// TwinCAT 3 PLC project FactoryIOLibrary
// Title: FactoryIO_Library
// Company: Privat
// Author: Entwickler
// ProjectVersion: 0.0.8
// Description: This library contains function blocks to control scenes in FactoryIO.
// ProgramVersion: 3.1.4026.24
// libraries:
//   Tc2_Standard, * (Beckhoff Automation GmbH)
//   Tc2_System, * (Beckhoff Automation GmbH)
//   Tc2_Utilities, * (Beckhoff Automation GmbH)
//   Tc3_Module, * (Beckhoff Automation GmbH)
// project tree:
//   DUTs/Communication/ADS/ ADSCommunicationInterface.TcDUT
//   DUTs/HMI/Header/ HMIHeader.TcDUT (not stored)
//   DUTs/HMI/MachineSection/ HMIMovementForkInterface.TcDUT, HMIMovementInterface.TcDUT, HMIRFIDControlInterface.TcDUT, HMIRFIDDataInterface.TcDUT, HMIRFIDInterface.TcDUT, HMIRFIDStatusInterface.TcDUT (not stored), HMIRuncontrolInterface.TcDUT, HMIWindowSwitch.TcDUT (not stored), HMIWorkpieceInterface.TcDUT (not stored), MachineSection.TcDUT (not stored), MachineSectionHMIInterface.TcDUT
//   DUTs/HMI/NumericalInput/ HMIButtonNumericalInputInterface.TcDUT (not stored), HMINumericalInputInterface.TcDUT, HMINumericalInputLineInterface.TcDUT (not stored)
//   DUTs/HMI/SettingLine/ HMIButtonSettingLineInterface.TcDUT (not stored), HMISettingLineInterface.TcDUT (not stored)
//   DUTs/OperatingMode/ ActionState.TcDUT (not stored), FaultWarningState.TcDUT, HMIActionState.TcDUT (not stored), HMIInterfaceOperatingMode.TcDUT, HMIToPLCOperatingMode.TcDUT, OperatingMode.TcDUT, OperatingModeHomeing.TcDUT (not stored), PLCToHMIOperatingMode.TcDUT
//   DUTs/PickPlace/ PickPlacePosition.TcDUT (not stored)
//   DUTs/PositingBar/ PositingBarAlignmentDirection.TcDUT
//   DUTs/RFID/ RFIDReadSerialnumberStates.TcDUT (not stored), RFIDReadWriteDataStates.TcDUT
//   DUTs/VisionSensor/ VisionSensorParttype.TcDUT
//   POUs/AnalogValueHandling/ FC_AnalogInputValueHandling.TcPOU (not stored), FC_AnalogOutputValueHandling.TcPOU
//   POUs/Aufzug/ FB_Elevator.TcPOU (not stored)
//   POUs/Communication/ADS/ FB_ADSCommunicationStatus.TcPOU
//   POUs/Emitter/ FB_Emitter.TcPOU (not stored)
//   POUs/Foerderband/ FB_Foerderband.TcPOU
//   POUs/HMI/ FB_HMIHeader.TcPOU, FC_InitializingSettingLines.TcPOU (not stored)
//   POUs/OperatingMode/ FB_OperatingMode.TcPOU
//   POUs/PickPlace/ FB_PickPlace_DigitalAnalog.TcPOU (not stored)
//   POUs/PositingBar/ FB_PositingBar.TcPOU (not stored)
//   POUs/Remover/ FB_Remover.TcPOU
//   POUs/RFID/ FB_RFID.TcPOU (not stored)
//   POUs/VisionSensor/ FB_VisionSensor.TcPOU (not stored)
//   POUs/Warehouse/ FB_StackerCrane_Analog.TcPOU, FB_StackerCrane_Numerical.TcPOU
//   Version/ Global_Version.TcGVL

// ---- DUTs/Communication/ADS/ADSCommunicationInterface.TcDUT
TYPE ADSCommunicationInterface :
STRUCT
	LocalAMSNetId	:	STRING;
	DeviceIpAddress	:	STRING;
	RuntimeStatus	:	STRING;
	HeartbeatPLC	:	BOOL;
	HeartbeatHMI	:	BOOL;
END_STRUCT
END_TYPE

// ---- DUTs/HMI/MachineSection/HMIMovementForkInterface.TcDUT
TYPE HMIMovementForkInterface :
STRUCT
	ForkMovementSettingLines	:	ARRAY [1..3] of HMISettingLineInterface;
END_STRUCT
END_TYPE

// ---- DUTs/HMI/MachineSection/HMIMovementInterface.TcDUT
TYPE HMIMovementInterface :
STRUCT
	MovementSettingLines	:	ARRAY [1..3] OF HMISettingLineInterface;
	NumericalInput	:	HMINumericalInputInterface;
END_STRUCT
END_TYPE

// ---- DUTs/HMI/MachineSection/HMIRFIDControlInterface.TcDUT
TYPE HMIRFIDControlInterface :
STRUCT
	ExecuteCommand	:	BOOL;
	SelectedCommand	:	WORD;
	SelectedMemoryIndex	:	WORD;
END_STRUCT
END_TYPE

// ---- DUTs/HMI/MachineSection/HMIRFIDDataInterface.TcDUT
TYPE HMIRFIDDataInterface :
STRUCT
	SingleReadValue	:	WORD;
	SingleWriteValue	:	WORD;
	AllReadData	:	ARRAY[0..127] OF WORD;
	AllWriteData	:	ARRAY[0..127] OF WORD;
END_STRUCT
END_TYPE

// ---- DUTs/HMI/MachineSection/HMIRFIDInterface.TcDUT
TYPE HMIRFIDInterface :
STRUCT
	RFIDStatus	:	HMIRFIDStatusInterface;
	RFIDControl	:	HMIRFIDControlInterface;
	RFIDData	:	HMIRFIDDataInterface;
END_STRUCT
END_TYPE

// ---- DUTs/HMI/MachineSection/HMIRuncontrolInterface.TcDUT
TYPE HMIRuncontrolInterface :
STRUCT
	RuncontrolSettingLines	:	ARRAY [1..3] of HMISettingLineInterface;
END_STRUCT
END_TYPE

// ---- DUTs/HMI/MachineSection/MachineSectionHMIInterface.TcDUT
TYPE MachineSectionHMIInterface :
STRUCT
	ActiveMachineSection : MachineSection;
	SelectedActor : INT;
	Movements : HMIMovementInterface;
	Forks : HMIMovementForkInterface;
	Runcontrols : HMIRuncontrolInterface;
	RFID : HMIRFIDInterface;
	Workpiece : HMIWorkpieceInterface;
END_STRUCT
END_TYPE

// ---- DUTs/HMI/NumericalInput/HMINumericalInputInterface.TcDUT
TYPE HMINumericalInputInterface :
STRUCT
	CaptionNumericalInput	:	STRING;
	IsVisibleNumericalInput	:	BOOL;
	ValueLinesNumericalInput	:	ARRAY[1..2] OF HMINumericalInputLineInterface;
	ButtonsNumericalInput	:	ARRAY[1..2] OF HMIButtonNumericalInputInterface;
END_STRUCT
END_TYPE

// ---- DUTs/OperatingMode/FaultWarningState.TcDUT
TYPE FaultWarningState :
STRUCT
	IsActive :	BOOL;
END_STRUCT
END_TYPE

// ---- DUTs/OperatingMode/HMIInterfaceOperatingMode.TcDUT
TYPE HMIInterfaceOperatingMode :
STRUCT
	PLCToHMI	:	PLCToHMIOperatingMode;
	HMIToPLC	:	HMIToPLCOperatingMode;
END_STRUCT
END_TYPE

// ---- DUTs/OperatingMode/HMIToPLCOperatingMode.TcDUT
TYPE HMIToPLCOperatingMode :
STRUCT
	Manuel	:	HMIActionState;
	Automatic	:	HMIActionState;
	AutomaticStart	:	HMIActionState;
	AutomaticStop	:	HMIActionState;
	AutomaticHome	:	HMIActionState;
	Quit	:	HMIActionState;
	Reset	:	HMIActionState;
END_STRUCT
END_TYPE

// ---- DUTs/OperatingMode/OperatingMode.TcDUT
TYPE OperatingMode :
STRUCT
	ManuelIsActive	:	BOOL;
	AutomaticIsActive	:	BOOL;
	EStop			:	ActionState;
	Fault			:	FaultWarningState;
	Warning			:	FaultWarningState;
	AutomaticStart	:	ActionState;
	AutomaticStop	:	ActionState;
	Reset	:	ActionState;
	Quit	:	ActionState;
	AutomaticHome	:	OperatingModeHomeing;
END_STRUCT
END_TYPE

// ---- DUTs/OperatingMode/PLCToHMIOperatingMode.TcDUT
TYPE PLCToHMIOperatingMode :
STRUCT
	Manuel	:	ActionState;
	Automatic	:	ActionState;
	AutomaticStart	:	ActionState;
	Automaticstop	:	ActionState;
	AutomaticHome	:	ActionState;
	Reset	:	ActionState;
	Quit	:	ActionState;
	Fault	:	ActionState;
	
END_STRUCT
END_TYPE

// ---- DUTs/PositingBar/PositingBarAlignmentDirection.TcDUT
{attribute 'qualified_only'}
{attribute 'strict'}
{attribute 'to_string'}
TYPE PositingBarAlignmentDirection :
(
	AlingmentLeft := 0,
	AlingmentRight
);
END_TYPE

// ---- DUTs/RFID/RFIDReadWriteDataStates.TcDUT
{attribute 'qualified_only'}
{attribute 'strict'}
{attribute 'to_string'}
TYPE RFIDReadWriteDataStates :
(
	WAITINGTRIGGER := 0,
	SETTRIGGER,
	WAITINGRESPONSE,
	RESPONSE,
	ERRORACTIVE,
	FINISHED
);
END_TYPE

// ---- DUTs/VisionSensor/VisionSensorParttype.TcDUT
{attribute 'qualified_only'}
{attribute 'strict'}
{attribute 'to_string'}
TYPE VisionSensorParttype :
(
	None := 0,
	BlueRawMaterial,
	BlueProductLid,
	BlueProductBase,
	GreenRawMaterial,
	GreenProductLid,
	GreenProductBase,
	MetalRawMaterial,
	MetalProductLid,
	MetalProductBase,
	NotDectedable := 100
);
END_TYPE

// ---- Version/Global_Version.TcGVL
{attribute 'TcGenerated'}
{attribute 'no-analysis'}
{attribute 'linkalways'}
// This function has been automatically generated from the project information.
VAR_GLOBAL CONSTANT
	{attribute 'const_non_replaced'}
	stLibVersion_FactoryIO_Library : ST_LibVersion := (iMajor := 0, iMinor := 0, iBuild := 8, iRevision := 0, nFlags := 0, sVersion := '0.0.8');
END_VAR

// ---- POUs/AnalogValueHandling/FC_AnalogOutputValueHandling.TcPOU
FUNCTION FC_AnalogOutputValueHandling
VAR_INPUT
	Setpoint	:	REAL;
	UpperLimit	:	REAL;
	LowerLimit	:	REAL;
END_VAR
VAR_OUTPUT
	ConvertedValue	:	WORD;
END_VAR
VAR
	tempCalculatedValue	:	REAL;
	tempConvertedValue	:	WORD;
	tempValueWithOffset	:	WORD;
END_VAR

tempCalculatedValue := Setpoint * 10.0/(UpperLimit - LowerLimit);
tempConvertedValue := TO_WORD(tempCalculatedValue * 10.0);
tempValueWithOffset := tempConvertedValue * 10;

ConvertedValue := tempValueWithOffset;

END_FUNCTION

// ---- POUs/Communication/ADS/FB_ADSCommunicationStatus.TcPOU
FUNCTION_BLOCK FB_ADSCommunicationStatus
VAR_INPUT
	Timeout	:	TIME := T#1S;
	TimeoutHMI	:	TIME := T#1S;
	LocalAdsPort	:	T_AmsPort := 851;
	HeartbeatHMI	:	BOOL;
END_VAR
VAR
	instReadLocalAMSNetId	:	FB_GetLocalAmsNetId;
	statExecuteReadingLocalAMSNetId	:	BOOL := TRUE;
	statBusyReadLocalAMSNetId	:	BOOL;
	statErrorReadLocalAMSNetId	:	BOOL;
	statErrorNumberReadLocalAMSNetId	:	UDINT;
	statReadLocalAMSNetId	:	T_AmsNetID;
	statReadLocalAMSNetIdSeprated	:	T_AmsNetIdArr;
	
	statGettingIpAddress	:	BOOL;
	statLocalIpAddress	:	STRING;
	
	instReadADSState	:	ADSRDSTATE;
	statExecuteReadingAdsState	:	BOOL;
	statBusyReadAdsState	:	BOOL;
	statErrorReadAdsState	:	BOOL;
	statErrorNumberAdsState	:	UDINT;
	statReadAdsState	:	UDINT;
	
	statConvertingAdsState	:	BOOL;
	statConvertedAdsState	:	STRING;
	
	instHearbeatEvaluationHMITrue	:	TON;
	instHearbeatEvaluationHMIFalse	:	TON;
	statErrorHeartbeatHMIToLongTrue	:	BOOL;
	statErrorHeartbeatHMIToLongFalse	:	BOOL;
	statHearbeatHMIIsKeepAlive	:	BOOL;
	
	instHearbeatPLCTrue	:	TON;
	statHeartbeatPLCTrue	:	BOOL;
	statHearbeatPLC	:	BOOL;
END_VAR

(*===================== Reading local AMSNetId =====================*)
instReadLocalAMSNetId(bExecute := statExecuteReadingLocalAMSNetId,
					  tTimeOut := Timeout,
					  bBusy => statBusyReadLocalAMSNetId,
					  bError => statErrorReadLocalAMSNetId,
					  nErrId => statErrorNumberReadLocalAMSNetId,
					  AddrString => statReadLocalAMSNetId,
					  AddrBytes => statReadLocalAMSNetIdSeprated);
					  
IF NOT statBusyReadLocalAMSNetId AND NOT statErrorReadLocalAMSNetId AND
	statExecuteReadingLocalAMSNetId THEN
	statExecuteReadingLocalAMSNetId := FALSE;
	statGettingIpAddress := TRUE;
	statExecuteReadingAdsState := TRUE;
END_IF

(*===================== Getting IP-Address =====================*)
IF statGettingIpAddress THEN
	statLocalIpAddress := GetDeviceIpAddress(statReadLocalAMSNetIdSeprated);
	statGettingIpAddress := FALSE;
END_IF

(*===================== Reading Ads state =====================*)
instReadADSState(NETID := statReadLocalAMSNetId,
				 PORT := LocalAdsPort,
				 RDSTATE := statExecuteReadingAdsState,
			     TMOUT := Timeout,
				 BUSY => statBusyReadAdsState,
				 ERR => statErrorReadAdsState,
				 ERRID => statErrorNumberAdsState,
				 ADSSTATE => statReadAdsState);
					  
IF NOT statBusyReadAdsState AND NOT statErrorReadAdsState AND
	statExecuteReadingAdsState THEN
	statExecuteReadingAdsState := FALSE;
	statConvertingAdsState := TRUE;
END_IF

(*===================== Converting Ads state =====================*)
IF statConvertingAdsState THEN
	statConvertedAdsState := ConvertRuntimestatusInString(statReadAdsState);
	statConvertingAdsState := FALSE;
END_IF

(*===================== Evaluating Heartbeat HMI =====================*)
instHearbeatEvaluationHMITrue(IN := HeartbeatHMI,
							  PT := TimeoutHMI,
							  Q => statErrorHeartbeatHMIToLongTrue);
instHearbeatEvaluationHMIFalse(IN := NOT HeartbeatHMI,
							  PT := TimeoutHMI,
							  Q => statErrorHeartbeatHMIToLongFalse);
							  

statHearbeatHMIIsKeepAlive := NOT statErrorHeartbeatHMIToLongTrue AND NOT statErrorHeartbeatHMIToLongFalse;

(*===================== Creating Heartbeat PLC =====================*)
instHearbeatPLCTrue(IN := NOT statHeartbeatPLCTrue,
					PT := TimeoutHMI,
					Q => statHeartbeatPLCTrue);
							  
IF statHeartbeatPLCTrue THEN
	statHearbeatPLC := NOT statHearbeatPLC;
END_IF

PROPERTY PUBLIC AdsState : String
GET
AdsState := statConvertedAdsState;
END_GET
END_PROPERTY

METHOD PRIVATE ConvertRuntimestatusInString : String
VAR_INPUT
	CurrentDeviceStatus 	: 	UDINT;
END_VAR
VAR
	tempConvertedDeviceStatus	:	STRING;
END_VAR
CASE CurrentDeviceStatus OF
	0:
		tempConvertedDeviceStatus := 'Invalid';
	1:
		tempConvertedDeviceStatus := 'Idle';
	2:
		tempConvertedDeviceStatus := 'Reset';
	3:
		tempConvertedDeviceStatus := 'Init';
	4:
		tempConvertedDeviceStatus := 'Start';
	5:
		tempConvertedDeviceStatus := 'Run';
	6:
		tempConvertedDeviceStatus := 'Stop';
	7:
		tempConvertedDeviceStatus := 'Save cfg';
	8:
		tempConvertedDeviceStatus := 'Load cfg';
	9:
		tempConvertedDeviceStatus := 'Power failure';
	10:
		tempConvertedDeviceStatus := 'Power good';
	11:
		tempConvertedDeviceStatus := 'Error';
	12:
		tempConvertedDeviceStatus := 'Shutdown';
	13:
		tempConvertedDeviceStatus := 'Suspend';
	14:
		tempConvertedDeviceStatus := 'Resume';
	15:
		tempConvertedDeviceStatus := 'Config';
	16:
		tempConvertedDeviceStatus := 'Reconfig';
	17:
		tempConvertedDeviceStatus := 'Stopping';
	18:
		tempConvertedDeviceStatus := 'Incompatible';
	19:
		tempConvertedDeviceStatus := 'Execption';
	ELSE
		tempConvertedDeviceStatus := 'Not defined in system';			
END_CASE

ConvertRuntimestatusInString := tempConvertedDeviceStatus;
END_METHOD

METHOD PRIVATE GetDeviceIpAddress : String
VAR_INPUT
	CurrentAMSNetId	:	T_AmsNetIdArr;
END_VAR
VAR
	tempRunCounter	:	INT;
	tempIpAddressConverted	:	STRING;
END_VAR
FOR tempRunCounter := 0 TO 3 DO
	tempIpAddressConverted := CONCAT(tempIpAddressConverted, BYTE_TO_STRING(CurrentAMSNetId[tempRunCounter]));
	IF tempRunCounter < 3 THEN
		tempIpAddressConverted := CONCAT(tempIpAddressConverted, '.');
	END_IF
END_FOR

GetDeviceIpAddress := tempIpAddressConverted;
END_METHOD

PROPERTY PUBLIC HMICommunicationIsActive : BOOL
GET
HMICommunicationIsActive := statHearbeatHMIIsKeepAlive;
END_GET
END_PROPERTY

PROPERTY PUBLIC LocalAMSNetId : String
GET
LocalAMSNetId := statReadLocalAMSNetId;
END_GET
END_PROPERTY

PROPERTY PUBLIC LocalIpAddress : String
GET
LocalIpAddress := statLocalIpAddress;
END_GET
END_PROPERTY

PROPERTY PUBLIC PLCHeartbeatHMICommunication : BOOL
GET
PLCHeartbeatHMICommunication := statHearbeatPLC;
END_GET
END_PROPERTY

END_FUNCTION_BLOCK

// ---- POUs/Foerderband/FB_Foerderband.TcPOU
FUNCTION_BLOCK FB_Foerderband
VAR_INPUT
	SensorInfeed	:	BOOL;	//Sensor am Band Einlauf
	SensorOutfeed	:	BOOL;	//Sensor am Band Auslauf
	MaximumTimeRuncontrol	:	TIME;	//Maximale Zeit bis Fehler Laufkontrolle aktiviert wird
END_VAR
VAR_OUTPUT
	MotorForward	:	BOOL;	//Motor vorwaerts drehen
	MotorBackward	:	BOOL;	//Motor rueckwaerts drehen
	RuncontrolForwardActive	:	BOOL;	//Laufkontrolle in Vorwaerts-Richtung aktiv
	RuncontrolBackwardActive	:	BOOL;	//Laufkontrolle in Rueckwaerts-Richtung aktiv
	Error	:	BOOL;	//Fehler aktiv
END_VAR
VAR_IN_OUT
	OperatingMode	:	OperatingMode;	//Schnittstelle für Betriebsarten
END_VAR
VAR
	statMotorForward	:	BOOL;
	statMotorBackward	:	BOOL;
	statRuncontrolForward	:	BOOL;
	statRuncontrolBackward	:	BOOL;
	statErrorRuncontrolForward	:	BOOL;
	statErrorRuncontrolBackward	:	BOOL;
	statTimeRuncontrolForward	:	TON;
	statTimeRuncontrolBackward	:	TON;
END_VAR

(*===================== Motor Forward =====================*)
statMotorForward := statMotorForward AND OperatingMode.AutomaticIsActive
									 AND(OperatingMode.AutomaticStart.IsActive OR 
										 OperatingMode.AutomaticHome.IsActive) AND NOT
										 statMotorBackward AND NOT
									 	 OperatingMode.AutomaticStop.IsActive AND NOT
									 	 OperatingMode.EStop.IsActive AND NOT
										 statErrorRuncontrolForward;
(*===================== Motor Backward =====================*)
statMotorBackward := statMotorBackward AND OperatingMode.AutomaticIsActive
									   AND(OperatingMode.AutomaticStart.IsActive OR 
										   OperatingMode.AutomaticHome.IsActive) AND NOT
										   statMotorForward AND NOT
									 	   OperatingMode.AutomaticStop.IsActive AND NOT
									 	   OperatingMode.EStop.IsActive AND NOT
										   statErrorRuncontrolBackward;
(*===================== Runcontrol Forward =====================*)
IF statMotorForward AND NOT statRuncontrolForward THEN
	statRuncontrolForward := TRUE;
ELSIF (statRuncontrolForward AND SensorOutfeed) OR
	(OperatingMode.Reset.IsActive AND statErrorRuncontrolForward)
THEN
		statRuncontrolForward := FALSE;
END_IF

statTimeRuncontrolForward(IN:= statRuncontrolForward,
						  PT:= MaximumTimeRuncontrol);
IF OperatingMode.Quit.IsActive THEN
	statErrorRuncontrolForward := FALSE;
END_IF
IF statTimeRuncontrolForward.Q THEN
	statErrorRuncontrolForward := TRUE;
END_IF
(*===================== Runcontrol Backward =====================*)
IF statMotorBackward AND NOT statRuncontrolBackward THEN
	statRuncontrolBackward := TRUE;
ELSIF statRuncontrolBackward AND SensorInfeed OR
	(OperatingMode.Reset.IsActive AND statErrorRuncontrolBackward)
THEN
		statRuncontrolBackward := FALSE;
END_IF

statTimeRuncontrolBackward(IN:= statRuncontrolBackward,
						   PT:= MaximumTimeRuncontrol);
IF OperatingMode.Quit.IsActive THEN
	statErrorRuncontrolBackward := FALSE;
END_IF
IF statTimeRuncontrolBackward.Q THEN
	statErrorRuncontrolBackward := TRUE;
END_IF
(*===================== Outputs =====================*)
MotorForward := statMotorForward;
MotorBackward := statMotorBackward;
RuncontrolForwardActive := statRuncontrolForward;
RuncontrolBackwardActive := statRuncontrolBackward;
Error := statErrorRuncontrolForward OR statErrorRuncontrolBackward;
OperatingMode.Fault.IsActive :=  statErrorRuncontrolForward OR statErrorRuncontrolBackward;

METHOD PUBLIC Motor_Off
VAR_INPUT
	Motor_Stop	:	BOOL;
END_VAR
IF Motor_Stop THEN
	statMotorForward := FALSE;
	statMotorBackward := FALSE;
END_IF
END_METHOD

METHOD MotorBackward_On
VAR_INPUT
	MotorBackward_Start	:	BOOL;
END_VAR
IF OperatingMode.AutomaticIsActive AND
(OperatingMode.AutomaticStart.IsActive OR 
 OperatingMode.AutomaticHome.IsActive) AND NOT
 statMotorForward AND NOT
 OperatingMode.AutomaticStop.IsActive AND NOT
 OperatingMode.EStop.IsActive AND NOT
 statErrorRuncontrolBackward AND NOT
 statMotorBackward AND
 MotorBackward_Start
 THEN
 	statMotorBackward := TRUE;
END_IF
END_METHOD

METHOD PUBLIC MotorForward_On
VAR_INPUT
	MotorForward_Start	:	BOOL;
END_VAR
IF  OperatingMode.AutomaticIsActive AND
(OperatingMode.AutomaticStart.IsActive OR 
 OperatingMode.AutomaticHome.IsActive) AND NOT
 statMotorBackward AND NOT
 OperatingMode.AutomaticStop.IsActive AND NOT
 OperatingMode.EStop.IsActive AND NOT
 statErrorRuncontrolForward AND NOT
 statMotorForward AND
 MotorForward_Start
 THEN
	statMotorForward := TRUE;
END_IF
END_METHOD

END_FUNCTION_BLOCK

// ---- POUs/HMI/FB_HMIHeader.TcPOU
FUNCTION_BLOCK FB_HMIHeader
VAR_INPUT
	NameApplication	:	STRING;
	OperatingModeHMIInterface	:	HMIInterfaceOperatingMode;
END_VAR
VAR_OUTPUT
END_VAR
VAR_IN_OUT
	HeaderHMIInterface	:	HMIHeader;
END_VAR
VAR
	statHeaderHMIInterface	:	HMIHeader;
END_VAR

(*===================== Name Application =====================*)
statHeaderHMIInterface.NameApplication := NameApplication;
(*===================== Name Application =====================*)
statHeaderHMIInterface.ErrorIsActive := OperatingModeHMIInterface.PLCToHMI.Fault.IsActive;
(*===================== Operating Mode =====================*)
IF OperatingModeHMIInterface.PLCToHMI.Manuel.IsActive THEN
	statHeaderHMIInterface.PathOperatingMode := 'Images/Manual_Mode.svg';
	statHeaderHMIInterface.State := 1;
ELSIF OperatingModeHMIInterface.PLCToHMI.Automatic.IsActive THEN
	statHeaderHMIInterface.PathOperatingMode := 'Images/Automatic_Mode.svg';
	statHeaderHMIInterface.State := 2;
END_IF
(*===================== Operating State =====================*)
IF OperatingModeHMIInterface.PLCToHMI.AutomaticStart.IsActive THEN
	statHeaderHMIInterface.PathMachineState := 'Images/Machine_Run.svg';
	statHeaderHMIInterface.State := 3;
ELSIF OperatingModeHMIInterface.PLCToHMI.AutomaticStop.IsActive THEN
	statHeaderHMIInterface.PathMachineState := 'Images/Machine_Stop.svg';
	statHeaderHMIInterface.State := 2;	
ELSIF OperatingModeHMIInterface.PLCToHMI.AutomaticHome.IsActive THEN
	statHeaderHMIInterface.PathMachineState := 'Images/Home-Symbol.svg';
	statHeaderHMIInterface.State := 4;			
END_IF
(*===================== Outputs =====================*)
HeaderHMIInterface := statHeaderHMIInterface;

END_FUNCTION_BLOCK

// ---- POUs/OperatingMode/FB_OperatingMode.TcPOU
FUNCTION_BLOCK FB_OperatingMode
VAR_INPUT
	PermissionHardware	:	BOOL;	//Permission hardware ready for operation
	PermissionSoftware	:	BOOL;	//Permission from safety machine ready for start
	E_Stop	:	BOOL;	//Button E-Stop
	OperatingModeManual	:	BOOL;	//Operating Mode manual is selected
	OperatingModeAutomatic	:	BOOL;	//Operating Mode automatic is selected
END_VAR
VAR_OUTPUT
	LEDStart	:	BOOL;	//Indicator to show state automatic start
	LEDStop	:	BOOL;	//Indicator to show state automatic stop
	LEDHome	:	BOOL;	//Indicator to show state automatic home
	LEDReset	:	BOOL;	//Indicator to show state reset
	LEDQuit	:	BOOL;	//Indicator to show state quit
END_VAR
VAR_IN_OUT
	HMIInterface	:	HMIInterfaceOperatingMode;
END_VAR
VAR
	statRisingEdgeAutomaticActivated	:	BOOL;	//Rising edge, used when Automatic is activated
	statOperatingMode	:	OperatingMode;
	statResetMethod	:	BOOL;
	statQuitMethod	:	BOOL;
	
	statHMIInterface	:	HMIInterfaceOperatingMode;
	statRisingEdgeManuelButtonPressedMachine	:	R_TRIG;
	statRisingEdgeManuelButtonPressedHMI	:	R_TRIG;
	statRisingEdgeAutomaticButtonPressedMachine	:	R_TRIG;
	statRisingEdgeAutomaticButtonPressedHMI	:	R_TRIG;
	statRisingEdgeAutomaticStartButtonPressedHMI	:	R_TRIG;
	statRisingEdgeAutomaticStopButtonPressedHMI	:	R_TRIG;
	statRisingEdgeAutomaticHomeButtonPressedHMI	:	R_TRIG;
END_VAR

(*===================== HMI-Interface umladen =====================*)
statHMIInterface := HMIInterface;
(*===================== Betriebsartenwahl =====================*)
statRisingEdgeManuelButtonPressedMachine(CLK := OperatingModeManual);
statRisingEdgeManuelButtonPressedHMI(CLK := statHMIInterface.HMIToPLC.Manuel.IsSelected);
statRisingEdgeAutomaticButtonPressedMachine(CLK := OperatingModeAutomatic);
statRisingEdgeAutomaticButtonPressedHMI(CLK := statHMIInterface.HMIToPLC.Automatic.IsSelected);
(*===================== Operating Manual =====================*)
statHMIInterface.PLCToHMI.Manuel.PreconditionsFullfilled := TRUE;
IF statRisingEdgeManuelButtonPressedMachine.Q OR
	(statRisingEdgeManuelButtonPressedHMI.Q AND statHMIInterface.PLCToHMI.Manuel.PreconditionsFullfilled)
	THEN
	statOperatingMode.ManuelIsActive := TRUE;
	statOperatingMode.AutomaticIsActive := FALSE;
END_IF
// statOperatingMode.ManuelIsActive := OperatingModeManual; 
(*===================== Operating Automatic =====================*)
statHMIInterface.PLCToHMI.Automatic.PreconditionsFullfilled := TRUE;
// statOperatingMode.AutomaticIsActive := OperatingModeAutomatic;
IF statRisingEdgeAutomaticButtonPressedMachine.Q OR
	(statRisingEdgeAutomaticButtonPressedHMI.Q AND statHMIInterface.PLCToHMI.Manuel.PreconditionsFullfilled)
	THEN
	statOperatingMode.AutomaticIsActive := TRUE;
	statOperatingMode.ManuelIsActive := FALSE;
END_IF
(*===================== HMI-Interface Betriebsarten =====================*)
statHMIInterface.PLCToHMI.Automatic.IsActive := statOperatingMode.AutomaticIsActive; 
statHMIInterface.PLCToHMI.Manuel.IsActive := statOperatingMode.ManuelIsActive;
(*===================== E-Stop is active =====================*)
statOperatingMode.EStop.PreconditionsFullfilled := TRUE;
statOperatingMode.EStop.IsActive := NOT E_Stop AND statOperatingMode.EStop.PreconditionsFullfilled;
(*===================== Reset is active =====================*)
statOperatingMode.Reset.PreconditionsFullfilled := TRUE;
statHMIInterface.PLCToHMI.Reset.PreconditionsFullfilled := statOperatingMode.Reset.PreconditionsFullfilled;
statOperatingMode.Reset.IsActive := (statResetMethod OR
									 statHMIInterface.HMIToPLC.Reset.IsSelected) AND 
									statOperatingMode.Reset.PreconditionsFullfilled;
statHMIInterface.PLCToHMI.Reset.IsActive := statOperatingMode.Reset.IsActive; 
(*===================== Quit is active =====================*)
statOperatingMode.Quit.PreconditionsFullfilled := TRUE;
statHMIInterface.PLCToHMI.Quit.PreconditionsFullfilled := statOperatingMode.Quit.PreconditionsFullfilled; 
statOperatingMode.Quit.IsActive := (statQuitMethod OR
									statHMIInterface.HMIToPLC.Quit.IsSelected) AND 
									statOperatingMode.Quit.PreconditionsFullfilled;
statHMIInterface.PLCToHMI.Quit.IsActive := statOperatingMode.Quit.IsActive; 
(*===================== Automatic Start is active =====================*)
statRisingEdgeAutomaticStartButtonPressedHMI(CLK := statHMIInterface.HMIToPLC.AutomaticStart.IsSelected);
statOperatingMode.AutomaticStart.PreconditionsFullfilled := PermissionHardware AND PermissionSoftware AND
												  			E_Stop AND NOT statOperatingMode.Reset.IsActive AND NOT
												  			statOperatingMode.AutomaticHome.IsActive AND NOT
															statOperatingMode.Fault.IsActive AND
												  			statOperatingMode.AutomaticIsActive;
statHMIInterface.PLCToHMI.AutomaticStart.PreconditionsFullfilled := statOperatingMode.AutomaticStart.PreconditionsFullfilled;
statOperatingMode.AutomaticStart.IsActive := (statOperatingMode.AutomaticStart.IsActive OR
											  statRisingEdgeAutomaticStartButtonPressedHMI.Q) AND
											  statOperatingMode.AutomaticStart.PreconditionsFullfilled;
IF statOperatingMode.AutomaticStart.IsActive AND statRisingEdgeAutomaticStartButtonPressedHMI.Q THEN
	statOperatingMode.AutomaticStop.IsActive := FALSE;
END_IF
statHMIInterface.PLCToHMI.AutomaticStart.IsActive := statOperatingMode.AutomaticStart.IsActive;
(*===================== Automatic Stop is active =====================*)
statRisingEdgeAutomaticStopButtonPressedHMI(CLK := statHMIInterface.HMIToPLC.AutomaticStop.IsSelected);
statOperatingMode.AutomaticStop.PreconditionsFullfilled := NOT statOperatingMode.AutomaticHome.IsActive;
statHMIInterface.PLCToHMI.AutomaticStop.PreconditionsFullfilled := statOperatingMode.AutomaticStop.PreconditionsFullfilled;
statOperatingMode.AutomaticStop.IsActive := ((statOperatingMode.AutomaticStop.IsActive OR statRisingEdgeAutomaticStopButtonPressedHMI.Q) AND
											 statOperatingMode.AutomaticStop.PreconditionsFullfilled) OR
											 statOperatingMode.ManuelIsActive OR statOperatingMode.Fault.IsActive OR 
											 (statOperatingMode.AutomaticIsActive AND (NOT PermissionHardware OR NOT PermissionSoftware)) OR
											  statOperatingMode.EStop.IsActive OR statOperatingMode.Reset.IsActive;
statHMIInterface.PLCToHMI.AutomaticStop.IsActive := statOperatingMode.AutomaticStop.IsActive;
IF statOperatingMode.AutomaticIsActive AND NOT statRisingEdgeAutomaticActivated THEN
	statRisingEdgeAutomaticActivated := TRUE;
	statOperatingMode.AutomaticStop.IsActive := TRUE;
ELSIF statOperatingMode.ManuelIsActive AND statRisingEdgeAutomaticActivated THEN
	statRisingEdgeAutomaticActivated := FALSE;
END_IF
IF statOperatingMode.AutomaticStop.IsActive AND statRisingEdgeAutomaticStopButtonPressedHMI.Q THEN
	statOperatingMode.AutomaticStop.IsActive := TRUE;
	statOperatingMode.AutomaticStart.IsActive := FALSE;
	statOperatingMode.AutomaticHome.IsActive := FALSE;
END_IF
(*===================== Automatic Home is active =====================*)
statRisingEdgeAutomaticHomeButtonPressedHMI(CLK := statHMIInterface.HMIToPLC.AutomaticHome.IsSelected);
statOperatingMode.AutomaticHome.IsReached := statOperatingMode.AutomaticHome.AllMachinesInHome;
IF statOperatingMode.AutomaticHome.IsReached THEN
	StateOperatingMode.AutomaticStop.IsActive := TRUE;
END_IF
statOperatingMode.AutomaticHome.PreconditionsFullfilled := PermissionHardware AND PermissionSoftware AND
												  			E_Stop AND NOT statOperatingMode.Reset.IsActive AND
												  			statOperatingMode.AutomaticIsActive AND NOT
														   statOperatingMode.AutomaticHome.IsReached;
statHMIInterface.PLCToHMI.AutomaticHome.PreconditionsFullfilled := statOperatingMode.AutomaticHome.PreconditionsFullfilled; 
statOperatingMode.AutomaticHome.IsActive := (statOperatingMode.AutomaticHome.IsActive OR
											statRisingEdgeAutomaticHomeButtonPressedHMI.Q) AND
											statOperatingMode.AutomaticHome.PreconditionsFullfilled;
IF statOperatingMode.AutomaticHome.IsActive AND statRisingEdgeAutomaticHomeButtonPressedHMI.Q THEN
	statOperatingMode.AutomaticHome.IsActive := TRUE;
	statOperatingMode.AutomaticStart.IsActive := FALSE;
	statOperatingMode.AutomaticStop.IsActive := FALSE;
END_IF
statHMIInterface.PLCToHMI.AutomaticHome.IsActive := statOperatingMode.AutomaticHome.IsActive; 
(*===================== Outputs =====================*)
LEDStart := statOperatingMode.AutomaticStart.IsActive;
LEDStop := statOperatingMode.AutomaticStop.IsActive;	
LEDHome := statOperatingMode.AutomaticHome.IsActive;	
LEDReset := statOperatingMode.Reset.IsActive;
LEDQuit	:= statOperatingMode.Quit.IsActive;
HMIInterface := statHMIInterface;

METHOD Homeing_On
VAR_INPUT
	ButtonHome	:	BOOL;
END_VAR
IF ButtonHome AND statOperatingMode.AutomaticStart.PreconditionsFullfilled AND NOT 
statOperatingMode.AutomaticHome.IsReached
THEN
	statOperatingMode.AutomaticStart.IsActive := FALSE;
	statOperatingMode.AutomaticStop.IsActive := FALSE;
	statOperatingMode.AutomaticHome.IsActive := TRUE;
END_IF
END_METHOD

METHOD PUBLIC Quit_On
VAR_INPUT
	ButtonQuit	:	BOOL;
END_VAR
IF ButtonQuit THEN
	statQuitMethod := TRUE;
ELSE
	statQuitMethod := FALSE;
END_IF
END_METHOD

METHOD PUBLIC Reset_on
VAR_INPUT
	ButtonReset	:	BOOL;
END_VAR
IF ButtonReset THEN
	statResetMethod := TRUE;
ELSE
	statResetMethod := FALSE;
END_IF
END_METHOD

METHOD PUBLIC Start_On
VAR_INPUT
	ButtonStart	:	BOOL;
END_VAR
IF ButtonStart AND statOperatingMode.AutomaticStart.PreconditionsFullfilled THEN
	statOperatingMode.AutomaticStart.IsActive := TRUE;
	statOperatingMode.AutomaticStop.IsActive := FALSE;
END_IF
END_METHOD

PROPERTY PUBLIC StateOperatingMode : REFERENCE TO OperatingMode
GET
StateOperatingMode REF= statOperatingMode;
END_GET
SET
statOperatingMode := StateOperatingMode;
END_SET
END_PROPERTY

METHOD PUBLIC Stop_On
VAR_INPUT
	ButtonStop	:	BOOL;
END_VAR
IF NOT ButtonStop AND statOperatingMode.AutomaticStart.PreconditionsFullfilled THEN
	statOperatingMode.AutomaticStart.IsActive := FALSE;
	statOperatingMode.AutomaticStop.IsActive := TRUE;
	statOperatingMode.AutomaticHome.IsActive := FALSE;
END_IF
END_METHOD

END_FUNCTION_BLOCK

// ---- POUs/Remover/FB_Remover.TcPOU
FUNCTION_BLOCK FB_Remover
VAR_INPUT
	PartPresent	:	BOOL;
	ActorInstanceIndex	:	INT;
	ActorInstanceName	:	STRING;
END_VAR
VAR_IN_OUT
	OperatingModeSection	:	OperatingMode;
	HMIInterface	:	MachineSectionHMIInterface;
END_VAR
VAR_OUTPUT
	RemovePart	:	BOOL;
END_VAR
VAR
	internRemovePart	: BOOL;
	internOperatingMode	:	OperatingMode;
	
	internHMIInterface	:	MachineSectionHMIInterface;
	internInstanceActivatedFirstTime	:	BOOL;
	internRisingEdgePressButton	:	R_TRIG;
END_VAR

(*===================== Operating mode =====================*)
internOperatingMode := OperatingModeSection;
(*===================== HMI Interface =====================*)
internHMIInterface := HMIInterface;

IF internHMIInterface.ActiveMachineSection = MachineSection.Remover AND
	internHMIInterface.SelectedActor = ActorInstanceIndex THEN
	(*===================== Initializing HMI-Interface =====================*)
	IF NOT internInstanceActivatedFirstTime THEN
		FC_InitializingSettingLines(HMIInterface := internHMIInterface);
		internInstanceActivatedFirstTime := TRUE;
	END_IF
	(*===================== Button Handling =====================*)
	internHMIInterface.Workpiece.WorkpieceSettingLines[1].CaptionSettingLine := CONCAT('Removing Part ', ActorInstanceName);
	internHMIInterface.Workpiece.WorkpieceSettingLines[1].VisibilitySettingLine := TRUE;
	
	internHMIInterface.Workpiece.WorkpieceSettingLines[1].SettingLineButtons[1].IsVisibleButton := TRUE;
	internHMIInterface.Workpiece.WorkpieceSettingLines[1].SettingLineButtons[1].IsVisibleAxisPosition := FALSE;
	internHMIInterface.Workpiece.WorkpieceSettingLines[1].SettingLineButtons[1].IsEnabled := PartPresent AND internOperatingMode.ManuelIsActive;
	internHMIInterface.Workpiece.WorkpieceSettingLines[1].SettingLineButtons[1].InPosition := NOT PartPresent;
	internHMIInterface.Workpiece.WorkpieceSettingLines[1].SettingLineButtons[1].CaptionButton := 'Remove';
	internHMIInterface.Workpiece.WorkpieceSettingLines[1].SettingLineButtons[1].PathImageButton := 'Images\RemovePartRemover.svg';
	
	internRisingEdgePressButton(CLK := internHMIInterface.Workpiece.WorkpieceSettingLines[1].SettingLineButtons[1].IsPressed);
	IF internRisingEdgePressButton.Q THEN
		internRemovePart := TRUE;
	END_IF
	(*===================== Write Interface =====================*)
	HMIInterface := internHMIInterface;
ELSE
		internInstanceActivatedFirstTime := FALSE;
END_IF
(*===================== Remove Parts =====================*)

IF NOT PartPresent THEN
	internRemovePart := FALSE;
END_IF

RemovePart := internRemovePart;

METHOD PUBLIC Remove : BOOL
IF PartPresent AND internOperatingMode.AutomaticIsActive AND
	internOperatingMode.AutomaticStart.IsActive
THEN
	internRemovePart := TRUE;
	Remove := TRUE;
ELSE
	Remove := FALSE;
END_IF
END_METHOD

END_FUNCTION_BLOCK

// ---- POUs/Warehouse/FB_StackerCrane_Analog.TcPOU
FUNCTION_BLOCK FB_StackerCrane_Analog
VAR_INPUT
	StackerCraneCurrentPositionXAxis	:	WORD;
	StackerCraneCurrentPositionZAxis	:	WORD;
	ActorInstanceIndex	:	INT;	//Index in DropDown HMI
	ActorInstanceName	:	STRING;		//Name of the instance
END_VAR
VAR_OUTPUT
	SetPointToXAxis : WORD;
	SetPointToZAxis : WORD;
	MoveForkLeft	:	BOOL;
	MoveForkRight	:	BOOL;
END_VAR
VAR_IN_OUT
	OperatingMode	:	OperatingMode;	//Schnittstelle für Betriebsarten
	HMIInterface	:	MachineSectionHMIInterface;	//HMI-Interface
END_VAR
VAR
	statMoveStackerCrane	:	BOOL;
	statStackerCraneInPositionXAxis	:	BOOL;
	statStackerCraneInPositionZAxis	:	BOOL;
	statMoveForkLeft	:	BOOL;
	statMoveForkRight	:	BOOL;
	statCurrentPositionXAxis	: REAL;
	statCurrentPositionZAxis	: REAL;
	statSelectedSetPointXAxis	: REAL;
	statSelectedSetPointZAxis	: REAL;
	statSetPointXAxis	:	REAL;
	statSetPointZAxis	:	REAL;
	statSetPointToXaxis	:	WORD;
	statSetPointToZaxis	:	WORD;
	
	internHMIInterface	:	MachineSectionHMIInterface;
	internInstanceActivatedFirstTime	:	BOOL;
	internRisingEdgePressButtonUpXAxis	:	R_TRIG;
	internRisingEdgePressButtonDownXAxis	:	R_TRIG;
	internRisingEdgePressButtonStopXAxis	:	R_TRIG;
	internRisingEdgePressButtonUpZAxis	:	R_TRIG;
	internRisingEdgePressButtonDownZAxis	:	R_TRIG;
	internRisingEdgePressButtonStopZAxis	:	R_TRIG;
	internRisingEdgePressButtonForkLeft	:	R_TRIG;
	internRisingEdgePressButtonForkRight	:	R_TRIG;
	internRisingEdgePressButtonMiddleFork	:	R_TRIG;
	internStopXAxis	:	BOOL;
	internStopZAxis	:	BOOL;
	internMiddleFork	:	BOOL;
END_VAR

(*===================== CurrentPosition Axes =====================*)
FC_AnalogInputValueHandling(RowValue:= StackerCraneCurrentPositionXAxis, 
							UpperLimit:= 10.5, 
							LowerLimit:= 0.0, 
							ConvertedValue=> statCurrentPositionXAxis);
FC_AnalogInputValueHandling(RowValue:= StackerCraneCurrentPositionZAxis, 
							UpperLimit:= 6.625, 
							LowerLimit:= 0.0, 
							ConvertedValue=> statCurrentPositionZAxis);
(*===================== HMI INTERFACE =====================*)
internHMIInterface := HMIInterface;

IF internHMIInterface.ActiveMachineSection = MachineSection.StackerCrane AND
	internHMIInterface.SelectedActor = ActorInstanceIndex THEN
	(*===================== Initializing HMI-Interface =====================*)
	IF NOT internInstanceActivatedFirstTime THEN
		FC_InitializingSettingLines(HMIInterface := internHMIInterface);
		internInstanceActivatedFirstTime := TRUE;
	END_IF
	(*===================== Button Handling Movement =====================*)
	internHMIInterface.Movements.MovementSettingLines[1].CaptionSettingLine := CONCAT('StackerCrane X-Axis Control ', ActorInstanceName);
	internHMIInterface.Movements.MovementSettingLines[1].VisibilitySettingLine := TRUE;
	
	internHMIInterface.Movements.MovementSettingLines[1].SettingLineButtons[1].IsVisibleButton := TRUE;
	internHMIInterface.Movements.MovementSettingLines[1].SettingLineButtons[1].IsVisibleAxisPosition := FALSE;
	internHMIInterface.Movements.MovementSettingLines[1].SettingLineButtons[1].IsEnabled := OperatingMode.ManuelIsActive AND NOT
									 														OperatingMode.EStop.IsActive AND NOT
																							OperatingMode.Fault.IsActive AND NOT
																							statMoveStackerCrane AND
																							statSetPointXAxis < 10.5;
	internHMIInterface.Movements.MovementSettingLines[1].SettingLineButtons[1].InPosition := statStackerCraneInPositionXAxis;
	internHMIInterface.Movements.MovementSettingLines[1].SettingLineButtons[1].CaptionButton := 'Right';
	internHMIInterface.Movements.MovementSettingLines[1].SettingLineButtons[1].PathImageButton := 'Images\ForwardConveyor.svg';
	
	internHMIInterface.Movements.MovementSettingLines[1].SettingLineButtons[2].IsVisibleButton := TRUE;
	internHMIInterface.Movements.MovementSettingLines[1].SettingLineButtons[2].IsVisibleAxisPosition := TRUE;
	internHMIInterface.Movements.MovementSettingLines[1].SettingLineButtons[2].IsEnabled := OperatingMode.ManuelIsActive;
	internHMIInterface.Movements.MovementSettingLines[1].SettingLineButtons[2].InPosition := NOT statMoveStackerCrane;
	internHMIInterface.Movements.MovementSettingLines[1].SettingLineButtons[2].AxisPosition := statCurrentPositionXAxis;
	internHMIInterface.Movements.MovementSettingLines[1].SettingLineButtons[2].CaptionButton := 'Stop';
	internHMIInterface.Movements.MovementSettingLines[1].SettingLineButtons[2].PathImageButton := 'Images\StopConveyor.svg';
	
	internHMIInterface.Movements.MovementSettingLines[1].SettingLineButtons[3].IsVisibleButton := TRUE;
	internHMIInterface.Movements.MovementSettingLines[1].SettingLineButtons[3].IsVisibleAxisPosition := FALSE;
	internHMIInterface.Movements.MovementSettingLines[1].SettingLineButtons[3].IsEnabled := OperatingMode.ManuelIsActive AND NOT
									 														OperatingMode.EStop.IsActive AND NOT
																							OperatingMode.Fault.IsActive AND NOT
																							statMoveStackerCrane AND
																							statSetPointXAxis > 0;
	internHMIInterface.Movements.MovementSettingLines[1].SettingLineButtons[3].InPosition := statStackerCraneInPositionXAxis;
	internHMIInterface.Movements.MovementSettingLines[1].SettingLineButtons[3].CaptionButton := 'Left';
	internHMIInterface.Movements.MovementSettingLines[1].SettingLineButtons[3].PathImageButton := 'Images\BackwardConveyor.svg';
	
	internHMIInterface.Movements.MovementSettingLines[2].CaptionSettingLine := CONCAT('StackerCrane Z-Axis Control ', ActorInstanceName);
	internHMIInterface.Movements.MovementSettingLines[2].VisibilitySettingLine := TRUE;
	
	internHMIInterface.Movements.MovementSettingLines[2].SettingLineButtons[1].IsVisibleButton := TRUE;
	internHMIInterface.Movements.MovementSettingLines[2].SettingLineButtons[1].IsVisibleAxisPosition := FALSE;
	internHMIInterface.Movements.MovementSettingLines[2].SettingLineButtons[1].IsEnabled := OperatingMode.ManuelIsActive AND NOT
									 														OperatingMode.EStop.IsActive AND NOT
																							OperatingMode.Fault.IsActive AND NOT
																							statMoveStackerCrane AND
																							statSetPointZAxis < 10.5;
	internHMIInterface.Movements.MovementSettingLines[2].SettingLineButtons[1].InPosition := statStackerCraneInPositionZAxis;
	internHMIInterface.Movements.MovementSettingLines[2].SettingLineButtons[1].CaptionButton := 'Up';
	internHMIInterface.Movements.MovementSettingLines[2].SettingLineButtons[1].PathImageButton := 'Images\UpElevator.svg';
	
	internHMIInterface.Movements.MovementSettingLines[2].SettingLineButtons[2].IsVisibleButton := TRUE;
	internHMIInterface.Movements.MovementSettingLines[2].SettingLineButtons[2].IsVisibleAxisPosition := TRUE;
	internHMIInterface.Movements.MovementSettingLines[2].SettingLineButtons[2].IsEnabled := OperatingMode.ManuelIsActive;
	internHMIInterface.Movements.MovementSettingLines[2].SettingLineButtons[2].InPosition := NOT statMoveStackerCrane;
	internHMIInterface.Movements.MovementSettingLines[2].SettingLineButtons[2].AxisPosition := statCurrentPositionZAxis;
	internHMIInterface.Movements.MovementSettingLines[2].SettingLineButtons[2].CaptionButton := 'Stop';
	internHMIInterface.Movements.MovementSettingLines[2].SettingLineButtons[2].PathImageButton := 'Images\StopConveyor.svg';
	
	internHMIInterface.Movements.MovementSettingLines[2].SettingLineButtons[3].IsVisibleButton := TRUE;
	internHMIInterface.Movements.MovementSettingLines[2].SettingLineButtons[3].IsVisibleAxisPosition := FALSE;
	internHMIInterface.Movements.MovementSettingLines[2].SettingLineButtons[3].IsEnabled := OperatingMode.ManuelIsActive AND NOT
									 														OperatingMode.EStop.IsActive AND NOT
																							OperatingMode.Fault.IsActive AND NOT
																							statMoveStackerCrane AND
																							statSetPointZAxis > 0;
	internHMIInterface.Movements.MovementSettingLines[2].SettingLineButtons[3].InPosition := statStackerCraneInPositionXAxis;
	internHMIInterface.Movements.MovementSettingLines[2].SettingLineButtons[3].CaptionButton := 'Down';
	internHMIInterface.Movements.MovementSettingLines[2].SettingLineButtons[3].PathImageButton := 'Images\DownElevator.svg';
	
	internHMIInterface.Forks.ForkMovementSettingLines[1].CaptionSettingLine := CONCAT('Fork Control ', ActorInstanceName);
	internHMIInterface.Forks.ForkMovementSettingLines[1].VisibilitySettingLine := TRUE;
	
	internHMIInterface.Forks.ForkMovementSettingLines[1].SettingLineButtons[1].IsVisibleButton := TRUE;
	internHMIInterface.Forks.ForkMovementSettingLines[1].SettingLineButtons[1].IsVisibleAxisPosition := FALSE;
	internHMIInterface.Forks.ForkMovementSettingLines[1].SettingLineButtons[1].IsEnabled := OperatingMode.ManuelIsActive AND NOT
									 														OperatingMode.EStop.IsActive AND NOT
																							OperatingMode.Fault.IsActive AND NOT
																							statMoveStackerCrane AND
																							statStackerCraneInPositionXAxis AND
																							statStackerCraneInPositionZAxis;
	internHMIInterface.Forks.ForkMovementSettingLines[1].SettingLineButtons[1].InPosition := statMoveForkLeft;
	internHMIInterface.Forks.ForkMovementSettingLines[1].SettingLineButtons[1].CaptionButton := 'Left';
	internHMIInterface.Forks.ForkMovementSettingLines[1].SettingLineButtons[1].PathImageButton := 'Images\BackwardConveyor.svg';
	
	internHMIInterface.Forks.ForkMovementSettingLines[1].SettingLineButtons[2].IsVisibleButton := TRUE;
	internHMIInterface.Forks.ForkMovementSettingLines[1].SettingLineButtons[2].IsVisibleAxisPosition := FALSE;
	internHMIInterface.Forks.ForkMovementSettingLines[1].SettingLineButtons[2].IsEnabled := OperatingMode.ManuelIsActive;
	internHMIInterface.Forks.ForkMovementSettingLines[1].SettingLineButtons[2].InPosition := NOT statMoveForkLeft AND NOT statMoveForkRight;
	internHMIInterface.Forks.ForkMovementSettingLines[1].SettingLineButtons[2].CaptionButton := 'Stop';
	internHMIInterface.Forks.ForkMovementSettingLines[1].SettingLineButtons[2].PathImageButton := 'Images\StopConveyor.svg';
	
	internHMIInterface.Forks.ForkMovementSettingLines[1].SettingLineButtons[3].IsVisibleButton := TRUE;
	internHMIInterface.Forks.ForkMovementSettingLines[1].SettingLineButtons[3].IsVisibleAxisPosition := FALSE;
	internHMIInterface.Forks.ForkMovementSettingLines[1].SettingLineButtons[3].IsEnabled := OperatingMode.ManuelIsActive AND NOT
									 														OperatingMode.EStop.IsActive AND NOT
																							OperatingMode.Fault.IsActive AND NOT
																							statMoveStackerCrane AND
																							statStackerCraneInPositionXAxis AND
																							statStackerCraneInPositionZAxis;
	internHMIInterface.Forks.ForkMovementSettingLines[1].SettingLineButtons[3].InPosition := statMoveForkRight;
	internHMIInterface.Forks.ForkMovementSettingLines[1].SettingLineButtons[3].CaptionButton := 'Right';
	internHMIInterface.Forks.ForkMovementSettingLines[1].SettingLineButtons[3].PathImageButton := 'Images\ForwardConveyor.svg';
	
	(*===================== X-Axis Up =====================*)
	internRisingEdgePressButtonUpXAxis(CLK := internHMIInterface.Movements.MovementSettingLines[1].SettingLineButtons[1].IsPressed);
	IF internRisingEdgePressButtonUpXAxis.Q THEN
		statSetPointXAxis := statSetPointXAxis + 0.2;
		statMoveStackerCrane := TRUE;
	END_IF
	(*===================== X-Axis Down =====================*)
	internRisingEdgePressButtonDownXAxis(CLK := internHMIInterface.Movements.MovementSettingLines[1].SettingLineButtons[3].IsPressed);
	IF internRisingEdgePressButtonDownXAxis.Q THEN
		statSetPointXAxis := statSetPointXAxis - 0.2;
		statMoveStackerCrane := TRUE;
	END_IF
	(*===================== X-Axis Stop =====================*)
	internRisingEdgePressButtonStopXAxis(CLK := internHMIInterface.Movements.MovementSettingLines[1].SettingLineButtons[2].IsPressed);
	IF internRisingEdgePressButtonStopXAxis.Q THEN
		internStopXAxis := TRUE;
	END_IF
	(*===================== Z-Axis Up =====================*)
	internRisingEdgePressButtonUpZAxis(CLK := internHMIInterface.Movements.MovementSettingLines[2].SettingLineButtons[1].IsPressed);
	IF internRisingEdgePressButtonUpZAxis.Q THEN
		statSetPointZAxis := statSetPointZAxis + 0.2;
		statMoveStackerCrane := TRUE;
	END_IF
	(*===================== Z-Axis Down =====================*)
	internRisingEdgePressButtonDownZAxis(CLK := internHMIInterface.Movements.MovementSettingLines[2].SettingLineButtons[3].IsPressed);
	IF internRisingEdgePressButtonDownZAxis.Q THEN
		statSetPointZAxis := statSetPointZAxis - 0.2;
		statMoveStackerCrane := TRUE;
	END_IF
	(*===================== Z-Axis Stop =====================*)
	internRisingEdgePressButtonStopZAxis(CLK := internHMIInterface.Movements.MovementSettingLines[2].SettingLineButtons[2].IsPressed);
	IF internRisingEdgePressButtonStopZAxis.Q THEN
		internStopZAxis := TRUE;
	END_IF
	(*===================== Fork Left =====================*)
	internRisingEdgePressButtonForkLeft(CLK := internHMIInterface.Forks.ForkMovementSettingLines[1].SettingLineButtons[1].IsPressed);
	IF internRisingEdgePressButtonForkLeft.Q THEN
		statMoveForkLeft := TRUE;
	END_IF
	(*===================== Fork Right =====================*)
	internRisingEdgePressButtonForkRight(CLK := internHMIInterface.Forks.ForkMovementSettingLines[1].SettingLineButtons[3].IsPressed);
	IF internRisingEdgePressButtonForkRight.Q THEN
		statMoveForkRight := TRUE;
	END_IF
	(*===================== Fork Middle =====================*)
	internRisingEdgePressButtonMiddleFork(CLK := internHMIInterface.Forks.ForkMovementSettingLines[1].SettingLineButtons[2].IsPressed);
	IF internRisingEdgePressButtonMiddleFork.Q THEN
		statMoveForkLeft := FALSE;
		statMoveForkRight := FALSE;
	END_IF
	
	(*===================== Write Interface =====================*)
	HMIInterface := internHMIInterface;
ELSE
		internInstanceActivatedFirstTime := FALSE;
END_IF
(*===================== Stacker crane in Position =====================*)
EvaluatePosition();
(*===================== Positioning Stacker crane =====================*)
IF ((OperatingMode.AutomaticIsActive AND OperatingMode.AutomaticStart.IsActive) OR
	(OperatingMode.ManuelIsActive)) 
   AND statMoveStackerCrane 
THEN
	statSelectedSetPointXAxis := statSetPointXAxis;
	statSelectedSetPointZAxis := statSetPointZAxis;
END_IF
IF OperatingMode.EStop.IsActive OR OperatingMode.Fault.IsActive OR 
((OperatingMode.AutomaticIsActive AND OperatingMode.AutomaticStop.IsActive) OR
(OperatingMode.ManuelIsActive AND (internStopXAxis OR internStopZAxis)))
THEN
	statSelectedSetPointXAxis := statCurrentPositionXAxis;
	statSelectedSetPointZAxis := statCurrentPositionZAxis;
	statMoveStackerCrane := FALSE;
END_IF
(*===================== SetPoint X-Axis =====================*)
FC_AnalogOutputValueHandling(Setpoint:= statSelectedSetPointXAxis, 
						     UpperLimit:= 10.5, 
							 LowerLimit:= 0.0, 
							 ConvertedValue=> statSetPointToXaxis);
(*===================== SetPoint Z-Axis =====================*)
FC_AnalogOutputValueHandling(Setpoint:= statSelectedSetPointZAxis, 
						     UpperLimit:= 6.625, 
							 LowerLimit:= 0.0, 
							 ConvertedValue=> statSetPointToZaxis);
(*===================== Outputs writting =====================*)
SetPointToXAxis := statSetPointToXaxis;
SetPointToZAxis := statSetPointToZaxis;
MoveForkLeft := statMoveForkLeft;
MoveForkRight := statMoveForkRight;

METHOD PUBLIC EvaluatePosition
IF statStackerCraneInPositionXAxis AND statStackerCraneInPositionZAxis THEN
	statMoveStackerCrane := FALSE;
END_IF
IF (statCurrentPositionXAxis >= statSetPointXAxis - 0.1) AND (statCurrentPositionXAxis <= statSetPointXAxis + 0.1) THEN
	statStackerCraneInPositionXAxis := TRUE;
ELSE
	statStackerCraneInPositionXAxis := FALSE;
END_IF
IF (statCurrentPositionZAxis >= statSetPointZAxis - 0.1) AND (statCurrentPositionZAxis <= statSetPointZAxis + 0.1) THEN
	statStackerCraneInPositionZAxis := TRUE;
ELSE
	statStackerCraneInPositionZAxis := FALSE;
END_IF
END_METHOD

PROPERTY PUBLIC InPositionXAxis : BOOL
GET
InPositionXAxis := statStackerCraneInPositionXAxis;
END_GET
END_PROPERTY

PROPERTY PUBLIC InPositionZAxis : BOOL
GET
InPositionZAxis := statStackerCraneInPositionZAxis;
END_GET
END_PROPERTY

METHOD PUBLIC MoveAxesStackerCrane_ON : BOOL
VAR_INPUT
	StartMoveStackerCrane	:	BOOL;
	PositionXAxis	:	REAL;
	PositionZAxis	:	REAL;
END_VAR
IF OperatingMode.AutomaticIsActive AND OperatingMode.AutomaticStart.IsActive AND
	NOT statMoveStackerCrane AND StartMoveStackerCrane THEN
	SetPointXAxis := PositionXAxis;
	SetPointZAxis := PositionZAxis;
	statMoveStackerCrane := TRUE;
// 	statStackerCraneInPositionXAxis := FALSE;
// 	statStackerCraneInPositionZAxis := FALSE;
END_IF
END_METHOD

METHOD PUBLIC MoveForkToLeft_ON : BOOL
VAR_INPUT
	StartMovingForkLeft	:	BOOL;
END_VAR
IF OperatingMode.AutomaticIsActive AND OperatingMode.AutomaticStart.IsActive AND
	InPositionXAxis AND InPositionZAxis AND StartMovingForkLeft AND NOT statMoveStackerCrane 
THEN
	statMoveForkLeft := TRUE;
	MoveForkToLeft_ON := TRUE;
ELSE
	MoveForkToLeft_ON := FALSE;
END_IF
END_METHOD

METHOD PUBLIC MoveForkToMiddle_ON : BOOL
VAR_INPUT
	StartMovingForkMiddle: BOOL;
END_VAR
IF OperatingMode.AutomaticIsActive AND OperatingMode.AutomaticStart.IsActive AND 
	StartMovingForkMiddle THEN
	statMoveForkLeft := FALSE;
	statMoveForkRight := FALSE;
	MoveForkToMiddle_ON := TRUE;
ELSE
	MoveForkToMiddle_ON := FALSE;
END_IF
END_METHOD

METHOD PUBLIC MoveForkToRight_ON : BOOL
VAR_INPUT
	StartMovingForkRight	:	BOOL;
END_VAR
IF OperatingMode.AutomaticIsActive AND OperatingMode.AutomaticStart.IsActive AND
	InPositionXAxis AND InPositionZAxis AND StartMovingForkRight  AND NOT statMoveStackerCrane
THEN
	statMoveForkRight := TRUE;
	MoveForkToRight_ON := TRUE;
ELSE
	MoveForkToRight_ON := FALSE;
END_IF
END_METHOD

PROPERTY PUBLIC SetPointXAxis : REAL
GET
SetPointXAxis := statSetPointXAxis;
END_GET
SET
IF SetPointXAxis < 10.5 THEN
	statSetPointXAxis := SetPointXAxis;
END_IF
END_SET
END_PROPERTY

PROPERTY PUBLIC SetPointZAxis : REAL
GET
SetPointZAxis := statSetPointZAxis;
END_GET
SET
IF SetPointZAxis < 6.125 THEN
	statSetPointZAxis := SetPointZAxis;	
END_IF
END_SET
END_PROPERTY

END_FUNCTION_BLOCK

// ---- POUs/Warehouse/FB_StackerCrane_Numerical.TcPOU
FUNCTION_BLOCK FB_StackerCrane_Numerical
VAR_INPUT
	XAxisMoving	:	BOOL;	//X axis is moving
	ZAxisMoving	:	BOOL;	//Z axis is moving
	ForkInPosLeft	:	BOOL;	//Fork is in the left position
	ForkInPosMiddle	:	BOOL;	//Fork is in the middle position
	ForkInPosRight	:	BOOL;	//Fork is in the right position
	ActorInstanceIndex	:	INT;	//Index in DropDown HMI
	ActorInstanceName	:	STRING;		//Name of the instance
END_VAR
VAR_OUTPUT
	LiftFork	:	BOOL;	//TRUE: Lift fork on current pos, FALSE: Lower fork on current pos, 
	MoveForkLeft	:	BOOL;	//Move Fork to the left pos
	MoveForkRight	:	BOOL;	//Move Fork to the right pos
	TargetPos	:	WORD;	//TargetPos for stacker crane
END_VAR
VAR_IN_OUT
	OperatingMode	:	OperatingMode;	//Schnittstelle für Betriebsarten
	HMIInterface	:	MachineSectionHMIInterface;	//HMI-Interface
END_VAR
VAR
	statMoveStackerCrane	:	BOOL;
	statStackerCraneNewOrder	:	BOOL;
	statStackerCraneInPositionXAxis	:	BOOL;
	statStackerCraneInPositionZAxis	:	BOOL;
	statMoveForkLeft	:	BOOL;
	statMoveForkRight	:	BOOL;
	statLiftFork	:	BOOL;
	statSelectedTargetPos	: WORD;
	statPropTargetPos	:	WORD;
	statREXAxisMoving	:	R_TRIG;
	statREZAxisMoving	:	R_TRIG;
	statFEXAxisMoving	:	F_TRIG;
	statFEZAxisMoving	:	F_TRIG;
	
	internHMIInterface	:	MachineSectionHMIInterface;
	internInstanceActivatedFirstTime	:	BOOL;
	internRisingEdgePressButtonConfirm	:	R_TRIG;
	internRisingEdgePressButtonMove	:	R_TRIG;
	internRisingEdgePressButtonForkLift	:	R_TRIG;
	internRisingEdgePressButtonForkLower	:	R_TRIG;
	internRisingEdgePressButtonForkLeft	:	R_TRIG;
	internRisingEdgePressButtonForkRight	:	R_TRIG;
	internRisingEdgePressButtonMiddleFork	:	R_TRIG;
	internMiddleFork	:	BOOL;
END_VAR

(*===================== HMI INTERFACE =====================*)
internHMIInterface := HMIInterface;

IF internHMIInterface.ActiveMachineSection = MachineSection.StackerCrane AND
	internHMIInterface.SelectedActor = ActorInstanceIndex THEN
	(*===================== Initializing HMI-Interface =====================*)
	IF NOT internInstanceActivatedFirstTime THEN
		FC_InitializingSettingLines(HMIInterface := internHMIInterface);
		internInstanceActivatedFirstTime := TRUE;
	END_IF
	(*===================== Button Handling Movement =====================*)
	internHMIInterface.Movements.NumericalInput.CaptionNumericalInput := 'Stacker Crane Target POS';
	internHMIInterface.Movements.NumericalInput.IsVisibleNumericalInput := TRUE;
	
	internHMIInterface.Movements.NumericalInput.ButtonsNumericalInput[1].IsVisibleButton := TRUE;
	internHMIInterface.Movements.NumericalInput.ButtonsNumericalInput[1].IsEnabled := OperatingMode.ManuelIsActive AND NOT
									 														OperatingMode.EStop.IsActive AND NOT
																							OperatingMode.Fault.IsActive AND NOT
																							statMoveStackerCrane;
	internHMIInterface.Movements.NumericalInput.ButtonsNumericalInput[1].InPosition := FALSE;
	internHMIInterface.Movements.NumericalInput.ButtonsNumericalInput[1].CaptionButton := 'Confirm';
	internHMIInterface.Movements.NumericalInput.ButtonsNumericalInput[1].PathImageButton := 'Images\ForwardConveyor.svg';
	
	internHMIInterface.Movements.NumericalInput.ButtonsNumericalInput[2].IsVisibleButton := TRUE;
	internHMIInterface.Movements.NumericalInput.ButtonsNumericalInput[2].IsEnabled := OperatingMode.ManuelIsActive;
	internHMIInterface.Movements.NumericalInput.ButtonsNumericalInput[2].InPosition := FALSE;
	internHMIInterface.Movements.NumericalInput.ButtonsNumericalInput[2].CaptionButton := 'Move';
	internHMIInterface.Movements.NumericalInput.ButtonsNumericalInput[2].PathImageButton := 'Images\StopConveyor.svg';
	
	internHMIInterface.Movements.NumericalInput.ValueLinesNumericalInput[1].CaptionDescription := 'Selected Pos:';
	internHMIInterface.Movements.NumericalInput.ValueLinesNumericalInput[1].UnitInput := 'Storage Place';
	internHMIInterface.Movements.NumericalInput.ValueLinesNumericalInput[1].IsEnabledInput := TRUE;
	
	internHMIInterface.Movements.NumericalInput.ValueLinesNumericalInput[2].CaptionDescription := 'Current Pos:';
	internHMIInterface.Movements.NumericalInput.ValueLinesNumericalInput[2].UnitInput := 'Storage Place';
	internHMIInterface.Movements.NumericalInput.ValueLinesNumericalInput[2].ValueInput := statSelectedTargetPos;
	internHMIInterface.Movements.NumericalInput.ValueLinesNumericalInput[2].IsEnabledInput := FALSE;
	
	internHMIInterface.Movements.MovementSettingLines[2].CaptionSettingLine := CONCAT('StackerCrane Lift function ', ActorInstanceName);
	internHMIInterface.Movements.MovementSettingLines[2].VisibilitySettingLine := TRUE;
	
	internHMIInterface.Movements.MovementSettingLines[2].SettingLineButtons[1].IsVisibleButton := TRUE;
	internHMIInterface.Movements.MovementSettingLines[2].SettingLineButtons[1].IsVisibleAxisPosition := FALSE;
	internHMIInterface.Movements.MovementSettingLines[2].SettingLineButtons[1].IsEnabled := OperatingMode.ManuelIsActive AND NOT
									 														OperatingMode.EStop.IsActive AND NOT
																							OperatingMode.Fault.IsActive AND NOT
																							statMoveStackerCrane;
	internHMIInterface.Movements.MovementSettingLines[2].SettingLineButtons[1].InPosition := FALSE;
	internHMIInterface.Movements.MovementSettingLines[2].SettingLineButtons[1].CaptionButton := 'Lift';
	internHMIInterface.Movements.MovementSettingLines[2].SettingLineButtons[1].PathImageButton := 'Images\UpElevator.svg';
	
	internHMIInterface.Movements.MovementSettingLines[2].SettingLineButtons[2].IsVisibleButton := TRUE;
	internHMIInterface.Movements.MovementSettingLines[2].SettingLineButtons[2].IsVisibleAxisPosition := FALSE;
	internHMIInterface.Movements.MovementSettingLines[2].SettingLineButtons[2].IsEnabled := OperatingMode.ManuelIsActive AND NOT
									 														OperatingMode.EStop.IsActive AND NOT
																							OperatingMode.Fault.IsActive AND NOT
																							statMoveStackerCrane;
	internHMIInterface.Movements.MovementSettingLines[2].SettingLineButtons[2].InPosition := FALSE;
	internHMIInterface.Movements.MovementSettingLines[2].SettingLineButtons[2].CaptionButton := 'Lower';
	internHMIInterface.Movements.MovementSettingLines[2].SettingLineButtons[2].PathImageButton := 'Images\DownElevator.svg';
	
	internHMIInterface.Forks.ForkMovementSettingLines[1].CaptionSettingLine := CONCAT('Fork Control ', ActorInstanceName);
	internHMIInterface.Forks.ForkMovementSettingLines[1].VisibilitySettingLine := TRUE;
	
	internHMIInterface.Forks.ForkMovementSettingLines[1].SettingLineButtons[1].IsVisibleButton := TRUE;
	internHMIInterface.Forks.ForkMovementSettingLines[1].SettingLineButtons[1].IsVisibleAxisPosition := FALSE;
	internHMIInterface.Forks.ForkMovementSettingLines[1].SettingLineButtons[1].IsEnabled := OperatingMode.ManuelIsActive AND NOT
									 														OperatingMode.EStop.IsActive AND NOT
																							OperatingMode.Fault.IsActive AND NOT
																							statMoveStackerCrane AND
																							statStackerCraneInPositionXAxis AND
																							statStackerCraneInPositionZAxis;
	internHMIInterface.Forks.ForkMovementSettingLines[1].SettingLineButtons[1].InPosition := statMoveForkLeft;
	internHMIInterface.Forks.ForkMovementSettingLines[1].SettingLineButtons[1].CaptionButton := 'Left';
	internHMIInterface.Forks.ForkMovementSettingLines[1].SettingLineButtons[1].PathImageButton := 'Images\BackwardConveyor.svg';
	
	internHMIInterface.Forks.ForkMovementSettingLines[1].SettingLineButtons[2].IsVisibleButton := TRUE;
	internHMIInterface.Forks.ForkMovementSettingLines[1].SettingLineButtons[2].IsVisibleAxisPosition := FALSE;
	internHMIInterface.Forks.ForkMovementSettingLines[1].SettingLineButtons[2].IsEnabled := OperatingMode.ManuelIsActive;
	internHMIInterface.Forks.ForkMovementSettingLines[1].SettingLineButtons[2].InPosition := NOT statMoveForkLeft AND NOT statMoveForkRight;
	internHMIInterface.Forks.ForkMovementSettingLines[1].SettingLineButtons[2].CaptionButton := 'Stop';
	internHMIInterface.Forks.ForkMovementSettingLines[1].SettingLineButtons[2].PathImageButton := 'Images\StopConveyor.svg';
	
	internHMIInterface.Forks.ForkMovementSettingLines[1].SettingLineButtons[3].IsVisibleButton := TRUE;
	internHMIInterface.Forks.ForkMovementSettingLines[1].SettingLineButtons[3].IsVisibleAxisPosition := FALSE;
	internHMIInterface.Forks.ForkMovementSettingLines[1].SettingLineButtons[3].IsEnabled := OperatingMode.ManuelIsActive AND NOT
									 														OperatingMode.EStop.IsActive AND NOT
																							OperatingMode.Fault.IsActive AND NOT
																							statMoveStackerCrane AND
																							statStackerCraneInPositionXAxis AND
																							statStackerCraneInPositionZAxis;
	internHMIInterface.Forks.ForkMovementSettingLines[1].SettingLineButtons[3].InPosition := statMoveForkRight;
	internHMIInterface.Forks.ForkMovementSettingLines[1].SettingLineButtons[3].CaptionButton := 'Right';
	internHMIInterface.Forks.ForkMovementSettingLines[1].SettingLineButtons[3].PathImageButton := 'Images\ForwardConveyor.svg';
	
	(*===================== Confirm =====================*)
	internRisingEdgePressButtonConfirm(CLK := internHMIInterface.Movements.NumericalInput.ButtonsNumericalInput[1].IsPressed);
	IF internRisingEdgePressButtonConfirm.Q THEN
		statPropTargetPos := REAL_TO_WORD(internHMIInterface.Movements.NumericalInput.ValueLinesNumericalInput[1].ValueInput);
	END_IF
	(*===================== Move =====================*)
	internRisingEdgePressButtonMove(CLK := internHMIInterface.Movements.NumericalInput.ButtonsNumericalInput[2].IsPressed);
	IF internRisingEdgePressButtonMove.Q THEN
		statMoveStackerCrane := TRUE;
		statStackerCraneNewOrder := TRUE;
	END_IF
	(*===================== Fork Lift =====================*)
	internRisingEdgePressButtonForkLift(CLK := internHMIInterface.Movements.MovementSettingLines[2].SettingLineButtons[1].IsPressed);
	IF internRisingEdgePressButtonForkLift.Q THEN
		statLiftFork := TRUE;
	END_IF
	(*===================== Fork Lower =====================*)
	internRisingEdgePressButtonForkLower(CLK := internHMIInterface.Movements.MovementSettingLines[2].SettingLineButtons[2].IsPressed);
	IF internRisingEdgePressButtonForkLower.Q THEN
		statLiftFork := FALSE;
	END_IF
	(*===================== Fork Left =====================*)
	internRisingEdgePressButtonForkLeft(CLK := internHMIInterface.Forks.ForkMovementSettingLines[1].SettingLineButtons[1].IsPressed);
	IF internRisingEdgePressButtonForkLeft.Q THEN
		statMoveForkLeft := TRUE;
	END_IF
	(*===================== Fork Right =====================*)
	internRisingEdgePressButtonForkRight(CLK := internHMIInterface.Forks.ForkMovementSettingLines[1].SettingLineButtons[3].IsPressed);
	IF internRisingEdgePressButtonForkRight.Q THEN
		statMoveForkRight := TRUE;
	END_IF
	(*===================== Fork Middle =====================*)
	internRisingEdgePressButtonMiddleFork(CLK := internHMIInterface.Forks.ForkMovementSettingLines[1].SettingLineButtons[2].IsPressed);
	IF internRisingEdgePressButtonMiddleFork.Q THEN
		statMoveForkLeft := FALSE;
		statMoveForkRight := FALSE;
	END_IF
	
	(*===================== Write Interface =====================*)
	HMIInterface := internHMIInterface;
ELSE
		internInstanceActivatedFirstTime := FALSE;
END_IF
(*===================== Stacker crane in Position =====================*)
statREXAxisMoving(CLK := XAxisMoving);
statFEXAxisMoving(CLK := XAxisMoving);
statREZAxisMoving(CLK := ZAxisMoving);
statFEZAxisMoving(CLK := ZAxisMoving);

IF statStackerCraneInPositionXAxis AND statStackerCraneInPositionZAxis AND
NOT statStackerCraneNewOrder
THEN
	statMoveStackerCrane := FALSE;
END_IF
IF statREXAxisMoving.Q THEN
	statStackerCraneInPositionXAxis := FALSE;
	statStackerCraneNewOrder := FALSE;
END_IF
IF statFEXAxisMoving.Q THEN
	statStackerCraneInPositionXAxis := TRUE;
END_IF
IF statREZAxisMoving.Q THEN
	statStackerCraneInPositionZAxis := FALSE;
	statStackerCraneNewOrder := FALSE;
END_IF
IF statFEZAxisMoving.Q THEN
	statStackerCraneInPositionZAxis := TRUE;
END_IF 
(*===================== Positioning Stacker crane =====================*)
IF ((OperatingMode.AutomaticIsActive AND OperatingMode.AutomaticStart.IsActive) OR
	(OperatingMode.ManuelIsActive)) 
   AND statMoveStackerCrane 
THEN
	statSelectedTargetPos := statPropTargetPos;
// 	statStackerCraneNewOrder := FALSE;
END_IF
IF OperatingMode.EStop.IsActive OR OperatingMode.Fault.IsActive OR 
OperatingMode.AutomaticIsActive AND OperatingMode.AutomaticStop.IsActive
THEN
	statSelectedTargetPos := 0;
	statMoveStackerCrane := FALSE;
END_IF
(*===================== Outputs writting =====================*)
LiftFork := statLiftFork;
MoveForkLeft := statMoveForkLeft;
MoveForkRight := statMoveForkRight;
TargetPos := statSelectedTargetPos;

PROPERTY PUBLIC InPositionXAxis : BOOL
GET
InPositionXAxis := statStackerCraneInPositionXAxis;
END_GET
END_PROPERTY

PROPERTY PUBLIC InPositionZAxis : BOOL
GET
InPositionZAxis := statStackerCraneInPositionZAxis;
END_GET
END_PROPERTY

METHOD PUBLIC LiftForkUp : BOOL
VAR_INPUT
	StartLiftingFork	:	BOOL;
END_VAR
IF OperatingMode.AutomaticIsActive AND OperatingMode.AutomaticStart.IsActive AND
	InPositionXAxis AND InPositionZAxis AND StartLiftingFork AND NOT statMoveStackerCrane 
THEN
	statLiftFork := TRUE;
	LiftForkUp := TRUE;
ELSE
	LiftForkUp := FALSE;
END_IF
END_METHOD

METHOD PUBLIC LowerForkUp : BOOL
VAR_INPUT
	StartLoweringFork	:	BOOL;
END_VAR
IF OperatingMode.AutomaticIsActive AND OperatingMode.AutomaticStart.IsActive AND
	InPositionXAxis AND InPositionZAxis AND StartLoweringFork AND NOT statMoveStackerCrane 
THEN
	statLiftFork := FALSE;
	LowerForkUp := TRUE;
ELSE
	LowerForkUp := FALSE;
END_IF
END_METHOD

METHOD PUBLIC MoveAxesStackerCrane_ON : BOOL
VAR_INPUT
	StartMoveStackerCrane	:	BOOL;
	TargetPosStackerCrane	:	WORD;
END_VAR
IF OperatingMode.AutomaticIsActive AND OperatingMode.AutomaticStart.IsActive AND
	NOT statMoveStackerCrane AND StartMoveStackerCrane AND 
NumericalTargetPos <> TargetPosStackerCrane 
THEN
	NumericalTargetPos := TargetPosStackerCrane;
	statMoveStackerCrane := TRUE;
	statStackerCraneNewOrder := TRUE;
END_IF
END_METHOD

METHOD PUBLIC MoveForkToLeft_ON : BOOL
VAR_INPUT
	StartMovingForkLeft	:	BOOL;
END_VAR
IF OperatingMode.AutomaticIsActive AND OperatingMode.AutomaticStart.IsActive AND
	InPositionXAxis AND InPositionZAxis AND StartMovingForkLeft AND NOT statMoveStackerCrane 
THEN
	statMoveForkLeft := TRUE;
	MoveForkToLeft_ON := TRUE;
ELSE
	MoveForkToLeft_ON := FALSE;
END_IF
END_METHOD

METHOD PUBLIC MoveForkToMiddle_ON : BOOL
VAR_INPUT
	StartMovingForkMiddle: BOOL;
END_VAR
IF OperatingMode.AutomaticIsActive AND OperatingMode.AutomaticStart.IsActive AND 
	StartMovingForkMiddle THEN
	statMoveForkLeft := FALSE;
	statMoveForkRight := FALSE;
	MoveForkToMiddle_ON := TRUE;
ELSE
	MoveForkToMiddle_ON := FALSE;
END_IF
END_METHOD

METHOD PUBLIC MoveForkToRight_ON : BOOL
VAR_INPUT
	StartMovingForkRight	:	BOOL;
END_VAR
IF OperatingMode.AutomaticIsActive AND OperatingMode.AutomaticStart.IsActive AND
	InPositionXAxis AND InPositionZAxis AND StartMovingForkRight  AND NOT statMoveStackerCrane
THEN
	statMoveForkRight := TRUE;
	MoveForkToRight_ON := TRUE;
ELSE
	MoveForkToRight_ON := FALSE;
END_IF
END_METHOD

PROPERTY PUBLIC NewOrderActive : BOOL
GET
NewOrderActive := statStackerCraneNewOrder;
END_GET
SET
statStackerCraneNewOrder := NewOrderActive;
END_SET
END_PROPERTY

PROPERTY PUBLIC NumericalTargetPos : WORD
GET
NumericalTargetPos := statPropTargetPos;
END_GET
SET
IF NumericalTargetPos > 0 AND NumericalTargetPos < 56 THEN
	statPropTargetPos := NumericalTargetPos;
END_IF
END_SET
END_PROPERTY

END_FUNCTION_BLOCK
